{attribute 'GeneratedUsingTerminal: EK1100-0000-0018'}
{attribute addProperty BoxType "EK1100-0000-0018"}
{attribute addProperty Id "Beckhoff_EL25xxEK1122Beckhoff_EL25xxEK1122_8334E3E72A_0001_EL2502_0000_0016EL2502_8962CF717A_0002_EL2502_0000_0017EL2502_8962CF717A_0003_EL2502_0000_0018EL2502_8962CF717A_0004_EL2502_0000_0019EL2502_8962CF717A_0005_EL2502_0000_0020EL2502_8962CF717A_0006_EL2502_0000_0021EL2502_8962CF717A_0007_EL2502_0000_0022EL2502_8962CF717A_0008_EL2502_0000_0023EL2502_8962CF717A_0009_EL2502_0000_0024EL2502_8962CF717A_0010_EL2502_0000_0025EL2502_8962CF717A_0011_EL2502_0000_0026EL2502_8962CF717A_0012_EL2502_0005_0016EL2502_8962CF717A_0013_EL2502_0010_0020EL2502_0F23744933A_0014_EL2521_0000_0000EL2521_336695F012A_0015_EL2521_0000_1016EL2521_3F36C7C828A_0016_EL2521_0000_1017EL2521_173EF27128A_0017_EL2521_0000_1018EL2521_173EF27128A_0018_EL2521_0000_1019EL2521_3513072828A_0019_EL2521_0000_1020EL2521_3513072828A_0020_EL2521_0000_1021EL2521_3513072828A_0021_EL2521_0000_1022EL2521_3513072828A_0022_EL2521_0024_1016EL2521_336695F012A_0023_EL2521_0024_1017EL2521_336695F012A_0024_EL2521_0024_1018EL2521_3513072828A_0025_EL2521_0024_1019EL2521_3513072828A_0026_EL2521_0024_1020EL2521_3513072828A_0027_EL2521_0024_1021EL2521_3513072828A_0028_EL2521_0025_1016EL2521_336695F012A_0029_EL2521_0025_1017EL2521_336695F012A_0030_EL2521_0025_1018EL2521_3513072828A_0031_EL2521_0025_1019EL2521_3513072828A_0032_EL2521_0025_1020EL2521_3513072828A_0033_EL2521_0025_1021EL2521_3513072828A_0034_EL2521_0124_0016EL2521_63978F5440A_0035_EL2521_0124_0017EL2521_63978F5440A_0036_EL2521_0124_0018EL2521_3637DCC642A_0037_EL2521_0124_0019EL2521_3637DCC642A_0038_EL2521_0124_0020EL2521_3637DCC642A_0039_EL2521_1001_0000EL2521_BF0777EB10A_0040_EL2521_1001_0001EL2521_336695F012A_0041_EL2521_1001_1016EL2521_336695F012A_0042_EL2521_1001_1017EL2521_336695F012A_0043_EL2521_1001_1018EL2521_3513072828A_0044_EL2521_1001_1019EL2521_3513072828A_0045_EL2521_1001_1020EL2521_3513072828A_0046_EL2522_0000_0017EL2522_CC50E1AE64A_0047_EL2522_0000_0018EL2522_CC50E1AE64A_0048_EL2522_0000_0021EL2522_CC50E1AE64A_0049_EL2522_0000_0022EL2522_CC50E1AE64A_0050_EL2535_0000_0016EL2535_2B2B792F24A_0051_EL2535_0000_0017EL2535_2B2B792F24A_0052_EL2535_0000_0018EL2535_2B2B792F24A_0053_EL2535_0000_0019EL2535_2B2B792F24A_0054_EL2535_0000_0021EL2535_2B2B792F24A_0055_EL2535_0000_0022EL2535_2B2B792F24A_0056_EL2535_0000_0023EL2535_2B2B792F24A_0057_EL2535_0002_0016EL2535_2B2B792F24A_0058_EL2535_0002_0017EL2535_2B2B792F24A_0059_EL2535_0002_0018EL2535_2B2B792F24A_0060_EL2535_0002_0019EL2535_2B2B792F24A_0061_EL2535_0002_0020EL2535_2B2B792F24A_0062_EL2535_0002_0021EL2535_2B2B792F24A_0063_EL2535_0002_0022EL2535_2B2B792F24A_0064_EL2535_0002_0023EL2535_2B2B792F24A_0065_EL2535_0005_0022EL2535_2B2B792F24A_0066_EL2535_0005_0023EL2535_2B2B792F24A_0067_EL2535_0050_0016EL2535_2B2B792F24A_0068_EL2535_0050_0017EL2535_2B2B792F24A_0069_EL2535_0050_0018EL2535_2B2B792F24A_0070_EL2535_0050_0019EL2535_2B2B792F24A_0071_EL2535_0050_0020EL2535_2B2B792F24A_0072_EL2535_0050_0021EL2535_2B2B792F24A_0073_EL2535_0050_0022EL2535_2B2B792F24A_0074_EL2535_0050_0023EL2535_2B2B792F24A_0075_EL2535_0100_0019EL2535_2B2B792F24A_0076_EL2535_0100_0020EL2535_2B2B792F24A_0077_EL2535_0100_0021EL2535_2B2B792F24A_0078_EL2535_0100_0022EL2535_2B2B792F24A_0079_EL2535_0100_0023EL2535_2B2B792F24A_0080_EL2535_0103_0023EL2535_2BC20E9122A_0081_EL2564_0000_0016EL2564_49D92DC824A_0082_EL2595_0000_0018EL2595_C979D21E13A_0083_EL2595_0000_0019EL2595_94B5C2E914A_0084_EL2596_0000_0017EL2596_5C974AD216A_0085_EL2596_0000_0018EL2596_5C974AD216A_0086_EL2596_0010_0016EL2596_5C974AD216"}
{attribute addProperty CRC "25772605"}
{attribute addProperty Size "2032"}
TYPE Beckhoff_EL25xx_0189423D EXTENDS EK1100_1FC0878B :
STRUCT
	{attribute addProperty Name "Beckhoff_EL25xxEK1122"}
	{attribute addProperty PreviousPort "Beckhoff EL25xx : B"}
	Beckhoff_EL25xxEK1122 : Beckhoff_EL25xxEK1122_8334E3E7;
	{attribute addProperty Name "A_0001_EL2502_0000_0016"}
	{attribute addProperty PreviousPort "Beckhoff EL25xxEK1122 : C"}
	A_0001_EL2502_0000_0016 : EL2502_8962CF71;
	{attribute addProperty Name "A_0002_EL2502_0000_0017"}
	{attribute addProperty PreviousPort "A_0001(EL2502-0000-0016) : B"}
	A_0002_EL2502_0000_0017 : EL2502_8962CF71;
	{attribute addProperty Name "A_0003_EL2502_0000_0018"}
	{attribute addProperty PreviousPort "A_0002(EL2502-0000-0017) : B"}
	A_0003_EL2502_0000_0018 : EL2502_8962CF71;
	{attribute addProperty Name "A_0004_EL2502_0000_0019"}
	{attribute addProperty PreviousPort "A_0003(EL2502-0000-0018) : B"}
	A_0004_EL2502_0000_0019 : EL2502_8962CF71;
	{attribute addProperty Name "A_0005_EL2502_0000_0020"}
	{attribute addProperty PreviousPort "A_0004(EL2502-0000-0019) : B"}
	A_0005_EL2502_0000_0020 : EL2502_8962CF71;
	{attribute addProperty Name "A_0006_EL2502_0000_0021"}
	{attribute addProperty PreviousPort "A_0005(EL2502-0000-0020) : B"}
	A_0006_EL2502_0000_0021 : EL2502_8962CF71;
	{attribute addProperty Name "A_0007_EL2502_0000_0022"}
	{attribute addProperty PreviousPort "A_0006(EL2502-0000-0021) : B"}
	A_0007_EL2502_0000_0022 : EL2502_8962CF71;
	{attribute addProperty Name "A_0008_EL2502_0000_0023"}
	{attribute addProperty PreviousPort "A_0007(EL2502-0000-0022) : B"}
	A_0008_EL2502_0000_0023 : EL2502_8962CF71;
	{attribute addProperty Name "A_0009_EL2502_0000_0024"}
	{attribute addProperty PreviousPort "A_0008(EL2502-0000-0023) : B"}
	A_0009_EL2502_0000_0024 : EL2502_8962CF71;
	{attribute addProperty Name "A_0010_EL2502_0000_0025"}
	{attribute addProperty PreviousPort "A_0009(EL2502-0000-0024) : B"}
	A_0010_EL2502_0000_0025 : EL2502_8962CF71;
	{attribute addProperty Name "A_0011_EL2502_0000_0026"}
	{attribute addProperty PreviousPort "A_0010(EL2502-0000-0025) : B"}
	A_0011_EL2502_0000_0026 : EL2502_8962CF71;
	{attribute addProperty Name "A_0012_EL2502_0005_0016"}
	{attribute addProperty PreviousPort "A_0011(EL2502-0000-0026) : B"}
	A_0012_EL2502_0005_0016 : EL2502_8962CF71;
	{attribute addProperty Name "A_0013_EL2502_0010_0020"}
	{attribute addProperty PreviousPort "A_0012(EL2502-0005-0016) : B"}
	A_0013_EL2502_0010_0020 : EL2502_0F237449;
	{attribute addProperty Name "A_0014_EL2521_0000_0000"}
	{attribute addProperty PreviousPort "A_0013(EL2502-0010-0020) : B"}
	A_0014_EL2521_0000_0000 : EL2521_336695F0;
	{attribute addProperty Name "A_0015_EL2521_0000_1016"}
	{attribute addProperty PreviousPort "A_0014(EL2521-0000-0000) : B"}
	A_0015_EL2521_0000_1016 : EL2521_3F36C7C8;
	{attribute addProperty Name "A_0016_EL2521_0000_1017"}
	{attribute addProperty PreviousPort "A_0015(EL2521-0000-1016) : B"}
	A_0016_EL2521_0000_1017 : EL2521_173EF271;
	{attribute addProperty Name "A_0017_EL2521_0000_1018"}
	{attribute addProperty PreviousPort "A_0016(EL2521-0000-1017) : B"}
	A_0017_EL2521_0000_1018 : EL2521_173EF271;
	{attribute addProperty Name "A_0018_EL2521_0000_1019"}
	{attribute addProperty PreviousPort "A_0017(EL2521-0000-1018) : B"}
	A_0018_EL2521_0000_1019 : EL2521_35130728;
	{attribute addProperty Name "A_0019_EL2521_0000_1020"}
	{attribute addProperty PreviousPort "A_0018(EL2521-0000-1019) : B"}
	A_0019_EL2521_0000_1020 : EL2521_35130728;
	{attribute addProperty Name "A_0020_EL2521_0000_1021"}
	{attribute addProperty PreviousPort "A_0019(EL2521-0000-1020) : B"}
	A_0020_EL2521_0000_1021 : EL2521_35130728;
	{attribute addProperty Name "A_0021_EL2521_0000_1022"}
	{attribute addProperty PreviousPort "A_0020(EL2521-0000-1021) : B"}
	A_0021_EL2521_0000_1022 : EL2521_35130728;
	{attribute addProperty Name "A_0022_EL2521_0024_1016"}
	{attribute addProperty PreviousPort "A_0021(EL2521-0000-1022) : B"}
	A_0022_EL2521_0024_1016 : EL2521_336695F0;
	{attribute addProperty Name "A_0023_EL2521_0024_1017"}
	{attribute addProperty PreviousPort "A_0022(EL2521-0024-1016) : B"}
	A_0023_EL2521_0024_1017 : EL2521_336695F0;
	{attribute addProperty Name "A_0024_EL2521_0024_1018"}
	{attribute addProperty PreviousPort "A_0023(EL2521-0024-1017) : B"}
	A_0024_EL2521_0024_1018 : EL2521_35130728;
	{attribute addProperty Name "A_0025_EL2521_0024_1019"}
	{attribute addProperty PreviousPort "A_0024(EL2521-0024-1018) : B"}
	A_0025_EL2521_0024_1019 : EL2521_35130728;
	{attribute addProperty Name "A_0026_EL2521_0024_1020"}
	{attribute addProperty PreviousPort "A_0025(EL2521-0024-1019) : B"}
	A_0026_EL2521_0024_1020 : EL2521_35130728;
	{attribute addProperty Name "A_0027_EL2521_0024_1021"}
	{attribute addProperty PreviousPort "A_0026(EL2521-0024-1020) : B"}
	A_0027_EL2521_0024_1021 : EL2521_35130728;
	{attribute addProperty Name "A_0028_EL2521_0025_1016"}
	{attribute addProperty PreviousPort "A_0027(EL2521-0024-1021) : B"}
	A_0028_EL2521_0025_1016 : EL2521_336695F0;
	{attribute addProperty Name "A_0029_EL2521_0025_1017"}
	{attribute addProperty PreviousPort "A_0028(EL2521-0025-1016) : B"}
	A_0029_EL2521_0025_1017 : EL2521_336695F0;
	{attribute addProperty Name "A_0030_EL2521_0025_1018"}
	{attribute addProperty PreviousPort "A_0029(EL2521-0025-1017) : B"}
	A_0030_EL2521_0025_1018 : EL2521_35130728;
	{attribute addProperty Name "A_0031_EL2521_0025_1019"}
	{attribute addProperty PreviousPort "A_0030(EL2521-0025-1018) : B"}
	A_0031_EL2521_0025_1019 : EL2521_35130728;
	{attribute addProperty Name "A_0032_EL2521_0025_1020"}
	{attribute addProperty PreviousPort "A_0031(EL2521-0025-1019) : B"}
	A_0032_EL2521_0025_1020 : EL2521_35130728;
	{attribute addProperty Name "A_0033_EL2521_0025_1021"}
	{attribute addProperty PreviousPort "A_0032(EL2521-0025-1020) : B"}
	A_0033_EL2521_0025_1021 : EL2521_35130728;
	{attribute addProperty Name "A_0034_EL2521_0124_0016"}
	{attribute addProperty PreviousPort "A_0033(EL2521-0025-1021) : B"}
	A_0034_EL2521_0124_0016 : EL2521_63978F54;
	{attribute addProperty Name "A_0035_EL2521_0124_0017"}
	{attribute addProperty PreviousPort "A_0034(EL2521-0124-0016) : B"}
	A_0035_EL2521_0124_0017 : EL2521_63978F54;
	{attribute addProperty Name "A_0036_EL2521_0124_0018"}
	{attribute addProperty PreviousPort "A_0035(EL2521-0124-0017) : B"}
	A_0036_EL2521_0124_0018 : EL2521_3637DCC6;
	{attribute addProperty Name "A_0037_EL2521_0124_0019"}
	{attribute addProperty PreviousPort "A_0036(EL2521-0124-0018) : B"}
	A_0037_EL2521_0124_0019 : EL2521_3637DCC6;
	{attribute addProperty Name "A_0038_EL2521_0124_0020"}
	{attribute addProperty PreviousPort "A_0037(EL2521-0124-0019) : B"}
	A_0038_EL2521_0124_0020 : EL2521_3637DCC6;
	{attribute addProperty Name "A_0039_EL2521_1001_0000"}
	{attribute addProperty PreviousPort "A_0038(EL2521-0124-0020) : B"}
	A_0039_EL2521_1001_0000 : EL2521_BF0777EB;
	{attribute addProperty Name "A_0040_EL2521_1001_0001"}
	{attribute addProperty PreviousPort "A_0039(EL2521-1001-0000) : B"}
	A_0040_EL2521_1001_0001 : EL2521_336695F0;
	{attribute addProperty Name "A_0041_EL2521_1001_1016"}
	{attribute addProperty PreviousPort "A_0040(EL2521-1001-0001) : B"}
	A_0041_EL2521_1001_1016 : EL2521_336695F0;
	{attribute addProperty Name "A_0042_EL2521_1001_1017"}
	{attribute addProperty PreviousPort "A_0041(EL2521-1001-1016) : B"}
	A_0042_EL2521_1001_1017 : EL2521_336695F0;
	{attribute addProperty Name "A_0043_EL2521_1001_1018"}
	{attribute addProperty PreviousPort "A_0042(EL2521-1001-1017) : B"}
	A_0043_EL2521_1001_1018 : EL2521_35130728;
	{attribute addProperty Name "A_0044_EL2521_1001_1019"}
	{attribute addProperty PreviousPort "A_0043(EL2521-1001-1018) : B"}
	A_0044_EL2521_1001_1019 : EL2521_35130728;
	{attribute addProperty Name "A_0045_EL2521_1001_1020"}
	{attribute addProperty PreviousPort "A_0044(EL2521-1001-1019) : B"}
	A_0045_EL2521_1001_1020 : EL2521_35130728;
	{attribute addProperty Name "A_0046_EL2522_0000_0017"}
	{attribute addProperty PreviousPort "A_0045(EL2521-1001-1020) : B"}
	A_0046_EL2522_0000_0017 : EL2522_CC50E1AE;
	{attribute addProperty Name "A_0047_EL2522_0000_0018"}
	{attribute addProperty PreviousPort "A_0046(EL2522-0000-0017) : B"}
	A_0047_EL2522_0000_0018 : EL2522_CC50E1AE;
	{attribute addProperty Name "A_0048_EL2522_0000_0021"}
	{attribute addProperty PreviousPort "A_0047(EL2522-0000-0018) : B"}
	A_0048_EL2522_0000_0021 : EL2522_CC50E1AE;
	{attribute addProperty Name "A_0049_EL2522_0000_0022"}
	{attribute addProperty PreviousPort "A_0048(EL2522-0000-0021) : B"}
	A_0049_EL2522_0000_0022 : EL2522_CC50E1AE;
	{attribute addProperty Name "A_0050_EL2535_0000_0016"}
	{attribute addProperty PreviousPort "A_0049(EL2522-0000-0022) : B"}
	A_0050_EL2535_0000_0016 : EL2535_2B2B792F;
	{attribute addProperty Name "A_0051_EL2535_0000_0017"}
	{attribute addProperty PreviousPort "A_0050(EL2535-0000-0016) : B"}
	A_0051_EL2535_0000_0017 : EL2535_2B2B792F;
	{attribute addProperty Name "A_0052_EL2535_0000_0018"}
	{attribute addProperty PreviousPort "A_0051(EL2535-0000-0017) : B"}
	A_0052_EL2535_0000_0018 : EL2535_2B2B792F;
	{attribute addProperty Name "A_0053_EL2535_0000_0019"}
	{attribute addProperty PreviousPort "A_0052(EL2535-0000-0018) : B"}
	A_0053_EL2535_0000_0019 : EL2535_2B2B792F;
	{attribute addProperty Name "A_0054_EL2535_0000_0021"}
	{attribute addProperty PreviousPort "A_0053(EL2535-0000-0019) : B"}
	A_0054_EL2535_0000_0021 : EL2535_2B2B792F;
	{attribute addProperty Name "A_0055_EL2535_0000_0022"}
	{attribute addProperty PreviousPort "A_0054(EL2535-0000-0021) : B"}
	A_0055_EL2535_0000_0022 : EL2535_2B2B792F;
	{attribute addProperty Name "A_0056_EL2535_0000_0023"}
	{attribute addProperty PreviousPort "A_0055(EL2535-0000-0022) : B"}
	A_0056_EL2535_0000_0023 : EL2535_2B2B792F;
	{attribute addProperty Name "A_0057_EL2535_0002_0016"}
	{attribute addProperty PreviousPort "A_0056(EL2535-0000-0023) : B"}
	A_0057_EL2535_0002_0016 : EL2535_2B2B792F;
	{attribute addProperty Name "A_0058_EL2535_0002_0017"}
	{attribute addProperty PreviousPort "A_0057(EL2535-0002-0016) : B"}
	A_0058_EL2535_0002_0017 : EL2535_2B2B792F;
	{attribute addProperty Name "A_0059_EL2535_0002_0018"}
	{attribute addProperty PreviousPort "A_0058(EL2535-0002-0017) : B"}
	A_0059_EL2535_0002_0018 : EL2535_2B2B792F;
	{attribute addProperty Name "A_0060_EL2535_0002_0019"}
	{attribute addProperty PreviousPort "A_0059(EL2535-0002-0018) : B"}
	A_0060_EL2535_0002_0019 : EL2535_2B2B792F;
	{attribute addProperty Name "A_0061_EL2535_0002_0020"}
	{attribute addProperty PreviousPort "A_0060(EL2535-0002-0019) : B"}
	A_0061_EL2535_0002_0020 : EL2535_2B2B792F;
	{attribute addProperty Name "A_0062_EL2535_0002_0021"}
	{attribute addProperty PreviousPort "A_0061(EL2535-0002-0020) : B"}
	A_0062_EL2535_0002_0021 : EL2535_2B2B792F;
	{attribute addProperty Name "A_0063_EL2535_0002_0022"}
	{attribute addProperty PreviousPort "A_0062(EL2535-0002-0021) : B"}
	A_0063_EL2535_0002_0022 : EL2535_2B2B792F;
	{attribute addProperty Name "A_0064_EL2535_0002_0023"}
	{attribute addProperty PreviousPort "A_0063(EL2535-0002-0022) : B"}
	A_0064_EL2535_0002_0023 : EL2535_2B2B792F;
	{attribute addProperty Name "A_0065_EL2535_0005_0022"}
	{attribute addProperty PreviousPort "A_0064(EL2535-0002-0023) : B"}
	A_0065_EL2535_0005_0022 : EL2535_2B2B792F;
	{attribute addProperty Name "A_0066_EL2535_0005_0023"}
	{attribute addProperty PreviousPort "A_0065(EL2535-0005-0022) : B"}
	A_0066_EL2535_0005_0023 : EL2535_2B2B792F;
	{attribute addProperty Name "A_0067_EL2535_0050_0016"}
	{attribute addProperty PreviousPort "A_0066(EL2535-0005-0023) : B"}
	A_0067_EL2535_0050_0016 : EL2535_2B2B792F;
	{attribute addProperty Name "A_0068_EL2535_0050_0017"}
	{attribute addProperty PreviousPort "A_0067(EL2535-0050-0016) : B"}
	A_0068_EL2535_0050_0017 : EL2535_2B2B792F;
	{attribute addProperty Name "A_0069_EL2535_0050_0018"}
	{attribute addProperty PreviousPort "A_0068(EL2535-0050-0017) : B"}
	A_0069_EL2535_0050_0018 : EL2535_2B2B792F;
	{attribute addProperty Name "A_0070_EL2535_0050_0019"}
	{attribute addProperty PreviousPort "A_0069(EL2535-0050-0018) : B"}
	A_0070_EL2535_0050_0019 : EL2535_2B2B792F;
	{attribute addProperty Name "A_0071_EL2535_0050_0020"}
	{attribute addProperty PreviousPort "A_0070(EL2535-0050-0019) : B"}
	A_0071_EL2535_0050_0020 : EL2535_2B2B792F;
	{attribute addProperty Name "A_0072_EL2535_0050_0021"}
	{attribute addProperty PreviousPort "A_0071(EL2535-0050-0020) : B"}
	A_0072_EL2535_0050_0021 : EL2535_2B2B792F;
	{attribute addProperty Name "A_0073_EL2535_0050_0022"}
	{attribute addProperty PreviousPort "A_0072(EL2535-0050-0021) : B"}
	A_0073_EL2535_0050_0022 : EL2535_2B2B792F;
	{attribute addProperty Name "A_0074_EL2535_0050_0023"}
	{attribute addProperty PreviousPort "A_0073(EL2535-0050-0022) : B"}
	A_0074_EL2535_0050_0023 : EL2535_2B2B792F;
	{attribute addProperty Name "A_0075_EL2535_0100_0019"}
	{attribute addProperty PreviousPort "A_0074(EL2535-0050-0023) : B"}
	A_0075_EL2535_0100_0019 : EL2535_2B2B792F;
	{attribute addProperty Name "A_0076_EL2535_0100_0020"}
	{attribute addProperty PreviousPort "A_0075(EL2535-0100-0019) : B"}
	A_0076_EL2535_0100_0020 : EL2535_2B2B792F;
	{attribute addProperty Name "A_0077_EL2535_0100_0021"}
	{attribute addProperty PreviousPort "A_0076(EL2535-0100-0020) : B"}
	A_0077_EL2535_0100_0021 : EL2535_2B2B792F;
	{attribute addProperty Name "A_0078_EL2535_0100_0022"}
	{attribute addProperty PreviousPort "A_0077(EL2535-0100-0021) : B"}
	A_0078_EL2535_0100_0022 : EL2535_2B2B792F;
	{attribute addProperty Name "A_0079_EL2535_0100_0023"}
	{attribute addProperty PreviousPort "A_0078(EL2535-0100-0022) : B"}
	A_0079_EL2535_0100_0023 : EL2535_2B2B792F;
	{attribute addProperty Name "A_0080_EL2535_0103_0023"}
	{attribute addProperty PreviousPort "A_0079(EL2535-0100-0023) : B"}
	A_0080_EL2535_0103_0023 : EL2535_2BC20E91;
	{attribute addProperty Name "A_0081_EL2564_0000_0016"}
	{attribute addProperty PreviousPort "A_0080(EL2535-0103-0023) : B"}
	A_0081_EL2564_0000_0016 : EL2564_49D92DC8;
	{attribute addProperty Name "A_0082_EL2595_0000_0018"}
	{attribute addProperty PreviousPort "A_0081(EL2564-0000-0016) : B"}
	A_0082_EL2595_0000_0018 : EL2595_C979D21E;
	{attribute addProperty Name "A_0083_EL2595_0000_0019"}
	{attribute addProperty PreviousPort "A_0082(EL2595-0000-0018) : B"}
	A_0083_EL2595_0000_0019 : EL2595_94B5C2E9;
	{attribute addProperty Name "A_0084_EL2596_0000_0017"}
	{attribute addProperty PreviousPort "A_0083(EL2595-0000-0019) : B"}
	A_0084_EL2596_0000_0017 : EL2596_5C974AD2;
	{attribute addProperty Name "A_0085_EL2596_0000_0018"}
	{attribute addProperty PreviousPort "A_0084(EL2596-0000-0017) : B"}
	A_0085_EL2596_0000_0018 : EL2596_5C974AD2;
	{attribute addProperty Name "A_0086_EL2596_0010_0016"}
	{attribute addProperty PreviousPort "A_0085(EL2596-0000-0018) : B"}
	A_0086_EL2596_0010_0016 : EL2596_5C974AD2;
END_STRUCT
END_TYPE

(* stored: Version 1.2.0.0, ProductVersion 3.1.4024.9
   DUT Beckhoff_EL25xx_0189423D: Id {39d88f4f-a373-432a-aa1e-467117612e50} *)
